{attribute 'GeneratedUsingTerminal: ELM3148-0000-0017'}
{attribute addProperty BoxType "ELM3148-0000-0017"}
{attribute addProperty Id "PAI_Status_Channel_1AT %I*PAI_Status_Channel_AE4AC1047PAI_Samples_1_Channel_1AT %I*PAI_Samples_1_Channel_EEA517254PAI_Timestamp_Channel_1AT %I*PAI_Timestamp_Channel_6DC4D2968PAI_Status_Channel_2AT %I*PAI_Status_Channel_AE4AC1047PAI_Samples_1_Channel_2AT %I*PAI_Samples_1_Channel_EEA517254PAI_Status_Channel_3AT %I*PAI_Status_Channel_AE4AC1047PAI_Samples_1_Channel_3AT %I*PAI_Samples_1_Channel_EEA517254PAI_Status_Channel_4AT %I*PAI_Status_Channel_AE4AC1047PAI_Samples_1_Channel_4AT %I*PAI_Samples_1_Channel_EEA517254PAI_Status_Channel_5AT %I*PAI_Status_Channel_AE4AC1047PAI_Samples_1_Channel_5AT %I*PAI_Samples_1_Channel_EEA517254PAI_Status_Channel_6AT %I*PAI_Status_Channel_AE4AC1047PAI_Samples_1_Channel_6AT %I*PAI_Samples_1_Channel_EEA517254PAI_Status_Channel_7AT %I*PAI_Status_Channel_AE4AC1047PAI_Samples_1_Channel_7AT %I*PAI_Samples_1_Channel_EEA517254PAI_Status_Channel_8AT %I*PAI_Status_Channel_AE4AC1047PAI_Samples_1_Channel_8AT %I*PAI_Samples_1_Channel_EEA517254WcStateAT %I*WcState_9091E0EB2InfoDataAT %I*InfoData_BEF6B88E18"}
{attribute addProperty CRC "137938472"}
{attribute addProperty Size "116"}
TYPE ELM3148_0838C628 EXTENDS EtcSlaveTerminalBase_947E5A46 :
STRUCT
	{attribute addProperty Name "PAI_Status_Channel_1"}
	PAI_Status_Channel_1 : PAI_Status_Channel_AE4AC104;
	{attribute addProperty Name "PAI_Samples_1_Channel_1"}
	PAI_Samples_1_Channel_1 : PAI_Samples_1_Channel_EEA51725;
	{attribute addProperty Name "PAI_Timestamp_Channel_1"}
	PAI_Timestamp_Channel_1 : PAI_Timestamp_Channel_6DC4D296;
	{attribute addProperty Name "PAI_Status_Channel_2"}
	PAI_Status_Channel_2 : PAI_Status_Channel_AE4AC104;
	{attribute addProperty Name "PAI_Samples_1_Channel_2"}
	PAI_Samples_1_Channel_2 : PAI_Samples_1_Channel_EEA51725;
	{attribute addProperty Name "PAI_Status_Channel_3"}
	PAI_Status_Channel_3 : PAI_Status_Channel_AE4AC104;
	{attribute addProperty Name "PAI_Samples_1_Channel_3"}
	PAI_Samples_1_Channel_3 : PAI_Samples_1_Channel_EEA51725;
	{attribute addProperty Name "PAI_Status_Channel_4"}
	PAI_Status_Channel_4 : PAI_Status_Channel_AE4AC104;
	{attribute addProperty Name "PAI_Samples_1_Channel_4"}
	PAI_Samples_1_Channel_4 : PAI_Samples_1_Channel_EEA51725;
	{attribute addProperty Name "PAI_Status_Channel_5"}
	PAI_Status_Channel_5 : PAI_Status_Channel_AE4AC104;
	{attribute addProperty Name "PAI_Samples_1_Channel_5"}
	PAI_Samples_1_Channel_5 : PAI_Samples_1_Channel_EEA51725;
	{attribute addProperty Name "PAI_Status_Channel_6"}
	PAI_Status_Channel_6 : PAI_Status_Channel_AE4AC104;
	{attribute addProperty Name "PAI_Samples_1_Channel_6"}
	PAI_Samples_1_Channel_6 : PAI_Samples_1_Channel_EEA51725;
	{attribute addProperty Name "PAI_Status_Channel_7"}
	PAI_Status_Channel_7 : PAI_Status_Channel_AE4AC104;
	{attribute addProperty Name "PAI_Samples_1_Channel_7"}
	PAI_Samples_1_Channel_7 : PAI_Samples_1_Channel_EEA51725;
	{attribute addProperty Name "PAI_Status_Channel_8"}
	PAI_Status_Channel_8 : PAI_Status_Channel_AE4AC104;
	{attribute addProperty Name "PAI_Samples_1_Channel_8"}
	PAI_Samples_1_Channel_8 : PAI_Samples_1_Channel_EEA51725;
	{attribute addProperty Name "WcState"}
	WcState : WcState_9091E0EB;
	{attribute addProperty Name "InfoData"}
	InfoData : InfoData_BEF6B88E;
END_STRUCT
END_TYPE

(* stored: Version 1.2.0.0, ProductVersion 3.1.4024.9
   DUT ELM3148_0838C628: Id {0a1be4b2-a6f9-4948-937c-42bcbde2b091} *)
